{attribute 'qualified_only'}
{attribute 'strict'}
TYPE E_TimeSource :
(
	FileTime := 0,
	DcTaskInfo := 1,
	fbLocalSystemTime := 2
);
END_TYPE

(* stored: Version 1.1.0.1, ProductVersion 3.1.4024.12
   DUT E_TimeSource: Id {562dee4f-bae0-4518-a8af-404a32355322} *)
